{attribute 'linkalways'} 
{attribute 'no_explicit_call' := 'This FB is a CLASS and must be accessed using methods or properties'}
{attribute 'enable_dynamic_creation'}
FUNCTION_BLOCK _TIME_OF_DAY EXTENDS DatatypeBase
VAR
	localData : TIME_OF_DAY;
	activeData : REFERENCE TO TIME_OF_DAY REF= localData;
END_VAR

PROPERTY PUBLIC Address : PVOID
GET
Address := ADR(activeData);
END_GET
END_PROPERTY

METHOD PUBLIC ClearReference
VAR_INPUT
END_VAR
activeData REF= localData;
END_METHOD

METHOD PUBLIC Clone : I_Datatype
VAR
    pClone : POINTER TO _TIME_OF_DAY;
END_VAR
pClone := __NEW(_TIME_OF_DAY(InitialValue := Value));
Clone := pClone^;
END_METHOD

METHOD FB_init : BOOL
VAR_INPUT
	bInitRetains : BOOL; // if TRUE, the retain variables are initialized (warm start / cold start)
	bInCopyCode : BOOL;  // if TRUE, the instance afterwards gets moved WORDo the copy code (online change)
	InitialValue : TIME_OF_DAY;
END_VAR
localData := InitialValue;
END_METHOD

PROPERTY PUBLIC IecType : T_MAXSTRING
GET
IecType := 'TIME_OF_DAY';
END_GET
END_PROPERTY

METHOD PUBLIC MakeReferenceTo
VAR_INPUT
	ReferenceTarget : REFERENCE TO TIME_OF_DAY;
END_VAR
activeData REF= ReferenceTarget;
END_METHOD

METHOD PUBLIC SerializeWith
VAR_INPUT
	Serializer : I_Serializer;
END_VAR
Serializer.AddTod(activeData);
END_METHOD

PROPERTY PUBLIC Size : UDINT
GET
Size := SIZEOF(activeData);
END_GET
END_PROPERTY

METHOD TryDeserializeFrom : BOOL
VAR_INPUT
	Deserializer : I_Deserializer;
END_VAR
TryDeserializeFrom := Deserializer.TryGetTod(activeData);
END_METHOD

METHOD TryMakeReferenceTo : BOOL
VAR_INPUT
	Target : I_Datatype;
END_VAR
VAR
	pTargetData : POINTER TO TIME_OF_DAY;
END_VAR
IF NOT (Target.IecType = IecType) THEN
	RETURN;
END_IF

pTargetData := Target.Address;
activeData REF= pTargetData^;
TryMakeReferenceTo := TRUE;
END_METHOD

PROPERTY PUBLIC Value : TIME_OF_DAY
GET
Value := activeData;
END_GET
SET
activeData := Value;
END_SET
END_PROPERTY

END_FUNCTION_BLOCK

(* stored: Version 1.1.0.1, ProductVersion 3.1.4024.12
   POU _TIME_OF_DAY: Id {2a5cbc79-5af0-024f-11d6-c106a4d218d8}, SpecialFunc None
   Folder Constructor: Id {b8553332-e89b-0e14-134b-4a990e9eaad4}
   Property Address: Id {e7076d61-8806-0a88-0e8e-82493ab2cb26}
   Get Get: Id {4354a89f-41ed-05ce-00a7-aa752f1d510b}
   Method ClearReference: Id {1a0a9a9b-3367-0a5e-369b-ba23186e5ddf}
   Method Clone: Id {af8952b2-1c27-0f71-1ee7-97b6d1d62e6e}
   Method FB_init: Id {6918d485-a7b6-0df0-382e-ed9b9ee1ea9d}
   Property IecType: Id {4d251238-7b32-0c3f-11d5-5dc080fadb33}
   Get Get: Id {38f8ea91-5cd2-0d74-10f0-4f5aff0833d6}
   Method MakeReferenceTo: Id {e6966efc-b41d-0643-200e-cf89b0301914}
   Method SerializeWith: Id {9d6bc285-569c-083e-33d5-12669a209112}
   Property Size: Id {70a4d714-eaff-00e2-00b2-21e191490afe}
   Get Get: Id {3c5e6d44-cc1a-0706-28bf-5b07ff078411}
   Method TryDeserializeFrom: Id {fe8effc3-f348-09b4-372e-1604ee3b8822}
   Method TryMakeReferenceTo: Id {a7cedc8d-f12b-0916-2998-cfdd5bed787f}
   Property Value: Id {cdf65d53-e5bc-071c-1b3f-201d8998d3f7}
   Get Get: Id {060e45eb-0c54-0c9f-28e0-2f1c3eebd0c1}
   Set Set: Id {498715c1-5c24-0ad8-3193-7356457f295d} *)
